{attribute 'pack_mode' := '0'}
TYPE ACMethodVacuumR EXTENDS ACMethodBaseR :
STRUCT
	//Ist-Druck
	_ActPressure : LREAL;
	//Dauer
	_ActDuration : TIME;
END_STRUCT
END_TYPE

(* stored: Version 1.1.0.1, ProductVersion 3.1.4020.12
   DUT ACMethodVacuumR: Id {57954b3e-440a-4a54-a592-5207b710ed6d} *)
